% RSLogix 500 project LAB 7 BWALTERS Ojohnson_BAK015.RSS, saved by version 8.40.00.08 %
PROJECT "UNTITLED"    % processor: MicroLogix 1400 %

PROGRAM FILES
  LAD 2   7 rungs

DATA FILES
  O0 OUTPUT  6 elements
  I1 INPUT  8 elements
  S2 STATUS  66 elements
  B3 BINARY  1 elements
  T4 TIMER  1 elements
  C5 COUNTER  6 elements
  R6 CONTROL  1 elements
  N7 INTEGER  1 elements
  F8 FLOAT  1 elements

LADDER 2
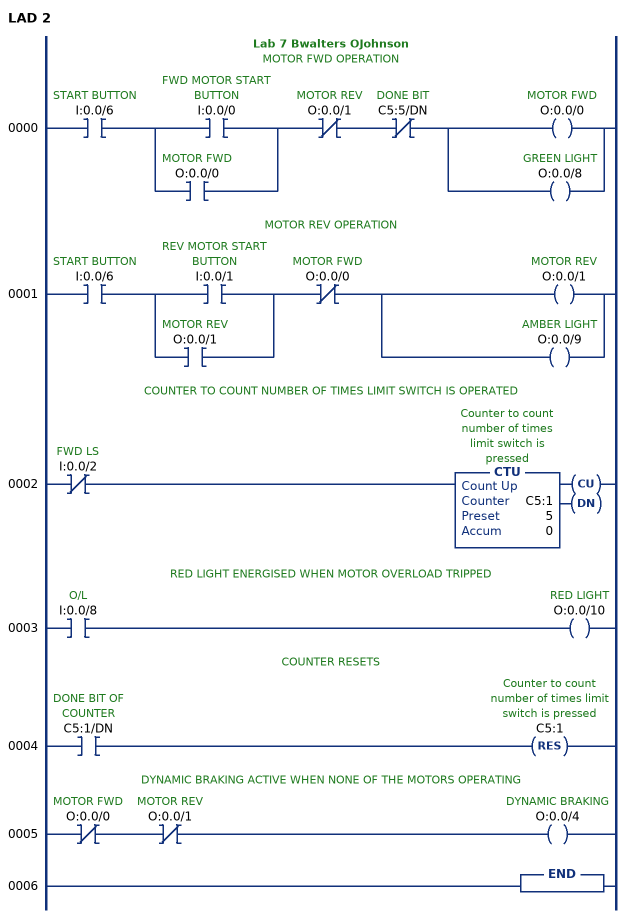
% Rung: 0 %
% TITLE: Lab 7 Bwalters OJohnson %
% MOTOR FWD OPERATION %
SOR XIC I:0.0/6 BST XIC I:0.0/0 NXB XIC O:0.0/0 BND XIO O:0.0/1 XIO C5:5/DN BST OTE O:0.0/0 NXB OTE O:0.0/8 BND EOR
%   I:0.0/6  "START BUTTON" %
%   I:0.0/0  "FWD MOTOR START BUTTON" %
%   O:0.0/0  "MOTOR FWD" %
%   O:0.0/1  "MOTOR REV" %
%   C5:5/DN  "DONE BIT" %
%   O:0.0/8  "GREEN LIGHT" %
% Rung: 1 %
% MOTOR REV OPERATION %
SOR XIC I:0.0/6 BST XIC I:0.0/1 NXB XIC O:0.0/1 BND XIO O:0.0/0 BST OTE O:0.0/1 NXB OTE O:0.0/9 BND EOR
%   I:0.0/6  "START BUTTON" %
%   I:0.0/1  "REV MOTOR START BUTTON" %
%   O:0.0/1  "MOTOR REV" %
%   O:0.0/0  "MOTOR FWD" %
%   O:0.0/9  "AMBER LIGHT" %
% Rung: 2 %
% COUNTER TO COUNT NUMBER OF TIMES LIMIT SWITCH IS OPERATED %
SOR XIO I:0.0/2 CTU C5:1 5 0 EOR
%   I:0.0/2  "FWD LS" %
%   C5:1  "Counter to count number of times limit switch is pressed" %
% Rung: 3 %
% RED LIGHT ENERGISED WHEN MOTOR OVERLOAD TRIPPED %
SOR XIC I:0.0/8 OTE O:0.0/10 EOR
%   I:0.0/8  "O/L" %
%   O:0.0/10  "RED LIGHT" %
% Rung: 4 %
% COUNTER RESETS %
SOR XIC C5:1/DN RES C5:1 EOR
%   C5:1/DN  "DONE BIT OF COUNTER" %
%   C5:1  "Counter to count number of times limit switch is pressed" %
% Rung: 5 %
% DYNAMIC BRAKING ACTIVE WHEN NONE OF THE MOTORS OPERATING %
SOR XIO O:0.0/0 XIO O:0.0/1 OTE O:0.0/4 EOR
%   O:0.0/0  "MOTOR FWD" %
%   O:0.0/1  "MOTOR REV" %
%   O:0.0/4  "DYNAMIC BRAKING" %
% Rung: 6 %
SOR END EOR

OTHER DOCUMENTED ADDRESSES
  I:0.0/5  "START"
  I:0.0/9  "FOWARD PUSH BUTTON"
  O:0.0/2  "MOTOR REV"

DATA TABLE (non-zero values as saved)
DATA C5
% .PRE .ACC %
% C5:1 % 5 0
